# EPICS autosave request: ADFireWireWin/firewireWinApp/Db/firewireDCAM_settings.req
$(P)$(R)FORMAT
$(P)$(R)MODE
$(P)$(R)FR
$(P)$(R)READOUT_TIME
